// TIA Portal V20 export
// export: Created 2025-12-01T14:57:09.4367768Z, ExportSetting None, DisplayName Totally Integrated Automation Portal, DisplayVersion V20 Update 3, DisplayName TIA Portal Openness, DisplayVersion V20 Update 3, DisplayName TIA Portal Version Control Interface, DisplayVersion V20 Update 3, DisplayName STEP 7 Professional, DisplayVersion V20 Update 3, DisplayName STEP 7 Safety, DisplayVersion V20 Update 2, DisplayName WinCC Basic/Comfort/Advanced, DisplayVersion V20 Update 3, DisplayName WinCC Professional, DisplayVersion V20 Update 3, DisplayName WinCC Unified, DisplayVersion V20 Update 3
FUNCTION "FC507_SIM_Ordenes_SRC_Clasificador" : Void   // FC507, LAD
{ S7_Optimized_Access := 'FALSE' }
AUTHOR : ROUTER
NAME : 20190911
VERSION : 3.1
// stored: AutoNumber false, SetENOAutomatically false
   VAR_INPUT
      Sacar_orden : Bool;
      Reset : Bool;
      Numero_Cruces : UDInt;   // MÁXIMO 15
   END_VAR
   VAR_OUTPUT
      Orden_FIFO : "ROUT_Orden_Fifo_Scanner";
   END_VAR
   VAR_IN_OUT
      Mem_FP : Bool;
      Aux_CNT : UDInt;
   END_VAR
   VAR_TEMP
      extraida : Bool;
      relleno : Byte;
      retval : Int;
      Suma_Bandejas_totales : UDInt;
      Bandejas_S3_menos1 : UDInt;
   END_VAR
   VAR_TEMP   // added for the SCL form of the ladder/FBD networks
      _w1 : Bool;
      _w2 : Bool;
      _w3 : Bool;
      _w4 : Bool;
   END_VAR
BEGIN

REGION Network 1
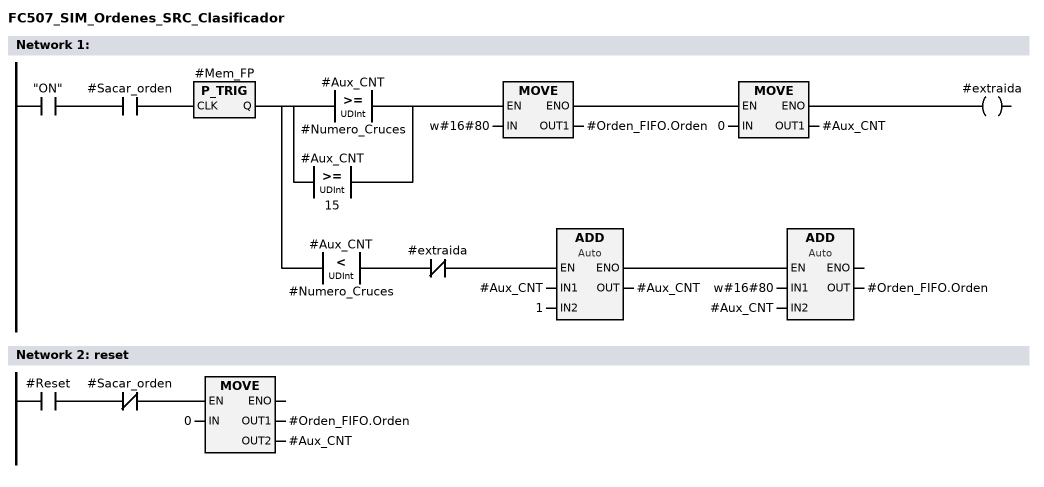
   RUNG wire#powerrail
      Contact( "ON" )
      Contact( #Sacar_orden )
      P_Trig( #Mem_FP )
      wire#w1
      { S7_Templates := "SrcType := UDInt" } GE_Contact(in1 := #Aux_CNT, in2 := #Numero_Cruces)
      wire#w2
      { S7_GenerateENO := "TRUE" } Move(in := w#16#80, out1 => #Orden_FIFO.Orden)
      { S7_GenerateENO := "TRUE" } Move(in := 0, out1 => #Aux_CNT)
      Coil( #extraida )
   END_RUNG
   RUNG wire#w1
      { S7_Templates := "SrcType := UDInt" } GE_Contact(in1 := #Aux_CNT, in2 := 15)
   END_RUNG wire#w2
   RUNG wire#w1
      { S7_Templates := "SrcType := UDInt" } LT_Contact(in1 := #Aux_CNT, in2 := #Numero_Cruces)
      I_Contact( #extraida )
      Add(in1 := #Aux_CNT, in2 := 1, out => #Aux_CNT)
      Add(in1 := w#16#80, in2 := #Aux_CNT, out => #Orden_FIFO.Orden)
   END_RUNG
   // the same network as SCL:
   // ENO of a box is taken as its EN; it also drops when the box reports an error
   #_w1 := "ON" AND #Sacar_orden;
   #_w2 := #_w1 AND NOT #Mem_FP;   // rising edge
   #Mem_FP := #_w1;
   #_w3 := #_w2 AND ((#Aux_CNT >= #Numero_Cruces) OR (#Aux_CNT >= 15));
   IF #_w3 THEN
       #Orden_FIFO.Orden := w#16#80;
       #Aux_CNT := 0;
   END_IF;
   #extraida := #_w3;
   #_w4 := #_w2 AND (#Aux_CNT < #Numero_Cruces) AND NOT #extraida;
   IF #_w4 THEN
       #Aux_CNT := #Aux_CNT + 1;
       #Orden_FIFO.Orden := w#16#80 + #Aux_CNT;
   END_IF;
END_REGION

REGION Network 2: reset
   RUNG wire#powerrail
      Contact( #Reset )
      I_Contact( #Sacar_orden )
      Move(in := 0, out1 => #Orden_FIFO.Orden, out2 => #Aux_CNT)
   END_RUNG
   // the same network as SCL:
   IF #Reset AND NOT #Sacar_orden THEN
       #Orden_FIFO.Orden := 0;
       #Aux_CNT := 0;
   END_IF;
END_REGION
END_FUNCTION
